// Mitsubishi GX Works2 project: 자기유지회로   PLC: Q02/Q02H

PROGRAM MAIN
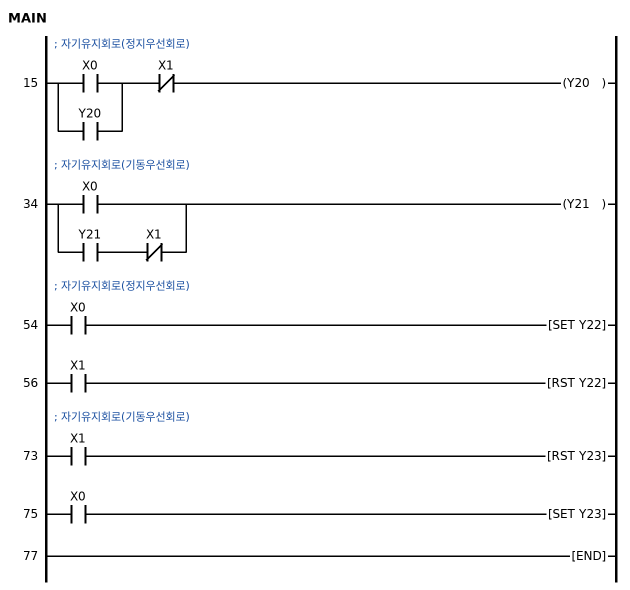
; 자기유지회로(정지우선회로)
15    LD      X0
      OR      Y20
      ANI     X1
      OUT     Y20
; 자기유지회로(기동우선회로)
34    LD      X0
      LD      Y21
      ANI     X1
      ORB
      OUT     Y21
; 자기유지회로(정지우선회로)
54    LD      X0
      SET     Y22
56    LD      X1
      RST     Y22
; 자기유지회로(기동우선회로)
73    LD      X1
      RST     Y23
75    LD      X0
      SET     Y23
77    END
END_PROGRAM
